VAR_GLOBAL CONSTANT
	
	g_mArmNum :INT := 2;	
	g_mJntNum :INT := 7;	
	g_sArmNum :INT := 4;	
	g_sJntNum :INT := 8;
	g_setupJntNum :INT :=5;
	g_cartDofs :INT :=6;
	g_cartJntNum:INT :=8;
	
	
	
	// control loop interval for each task
	g_slaveArmCtrlCycleTime :LREAL :=0.00025;
	g_slaveArmCtrlFreq :LREAL :=1.0/g_slaveArmCtrlCycleTime;
	g_armDynamicCycleTime :LREAL := 0.001;
	g_armDynamicFreq :LREAL := 1.0/g_armDynamicCycleTime;
	g_setupArmCtrlCycleTime :LREAL := 0.001;
	g_setupArmCtrlFreq :LREAL := 1.0/g_setupArmCtrlCycleTime;
	g_cartCtrlCycleTime :LREAL := 0.001;
	g_cartCtrlFreq :LREAL := 1.0/g_cartCtrlCycleTime;
	
	// wait time before robot init  for ethercat to stablize 
	g_robotInitWaitTime : LREAL := 1.0;

END_VAR

(* stored: Version 1.1.0.1, ProductVersion 3.1.4024.11
   GVL GVL_SystemParameters: Id {6ebbff17-e303-4344-870e-d2871229e24f} *)
